// TIA Portal V17 export
// export: Created 2023-04-07T13:41:58.3192772Z, ExportSetting WithDefaults, DisplayName Totally Integrated Automation Portal, DisplayVersion V17 Update 4, DisplayName TIA Portal Openness, DisplayVersion V17 Update 4, DisplayName TIA Portal Version Control Interface, DisplayVersion V17, DisplayName STEP 7 Professional, DisplayVersion V17 Update 4, DisplayName STEP 7 Safety, DisplayVersion V17, DisplayName WinCC Professional, DisplayVersion V17 Update 4
VAR_GLOBAL   // PLC tag table "Tabella delle variabili standard"
   "M12.0_Paolo" AT %M12.0 : Bool;
   "M12.1_Paolo" AT %M12.1 : Bool;
   System_Byte AT %MB1 : Byte;
   FirstScan AT %M1.0 : Bool;
   DiagStatusUpdate AT %M1.1 : Bool;
   AlwaysTRUE AT %M1.2 : Bool;
   AlwaysFALSE AT %M1.3 : Bool;
   Clock_Byte AT %MB0 : Byte;
   Clock_10Hz AT %M0.0 : Bool;
   Clock_5Hz AT %M0.1 : Bool;
   "Clock_2.5Hz" AT %M0.2 : Bool;
   Clock_2Hz AT %M0.3 : Bool;
   "Clock_1.25Hz" AT %M0.4 : Bool;
   Clock_1Hz AT %M0.5 : Bool;
   "Clock_0.625Hz" AT %M0.6 : Bool;
   "Clock_0.5Hz" AT %M0.7 : Bool;
   xDxP1 AT %M104.0 : Bool;
   xDxP2 AT %M104.1 : Bool;
   xDxP3 AT %M104.2 : Bool;
   xDxP4 AT %M104.3 : Bool;
   xSxP1 AT %M105.0 : Bool;
   xSxP2 AT %M105.1 : Bool;
   xSxP3 AT %M105.2 : Bool;
   xSxP4 AT %M105.3 : Bool;
   xPE1P1 AT %M106.0 : Bool;
   xPE1P2 AT %M106.1 : Bool;
   xPE1P3 AT %M106.2 : Bool;
   xPE1P4 AT %M106.3 : Bool;
   xMVSP1 AT %M107.0 : Bool;
   xMVSP2 AT %M107.1 : Bool;
   xMVSP3 AT %M107.2 : Bool;
   xMVSP4 AT %M107.3 : Bool;
   xPlcRun AT %M2.0 : Bool;
   xAlwaysOff AT %M20.0 : Bool;
   xPEP1 AT %M108.0 : Bool;
   xPEP2 AT %M108.1 : Bool;
   xPEP3 AT %M108.2 : Bool;
   xPEP4 AT %M108.3 : Bool;
   xSM1P1 AT %M109.0 : Bool;
   xSM1P2 AT %M109.1 : Bool;
   xSM2P1 AT %M109.4 : Bool;
   xSM2P2 AT %M109.5 : Bool;
   xAckPS AT %M110.0 : Bool;
   xPE10P1 AT %M106.4 : Bool;
   xPE10P2 AT %M106.5 : Bool;
   xPE10P3 AT %M106.6 : Bool;
   xPE10P4 AT %M106.7 : Bool;
   xDx10P1 AT %M104.4 : Bool;
   xDx10P2 AT %M104.5 : Bool;
   xDx10P3 AT %M104.6 : Bool;
   xDx10P4 AT %M104.7 : Bool;
   xSx10P1 AT %M105.4 : Bool;
   xSx10P2 AT %M105.5 : Bool;
   xSx10P3 AT %M105.6 : Bool;
   xSx10P4 AT %M105.7 : Bool;
   xFPlocal AT %M110.4 : Bool;
   xPEP11 AT %M108.4 : Bool;
   xPEP21 AT %M108.5 : Bool;
   xPEP31 AT %M108.6 : Bool;
   xPEP41 AT %M108.7 : Bool;
   xFNlocal AT %M110.5 : Bool;
   xDPCATL1 AT %M120.0 : Bool;
   xDPCATL2 AT %M120.1 : Bool;
   xMVSP11 AT %M107.4 : Bool;
   xMVSP21 AT %M107.5 : Bool;
   xMVSP31 AT %M107.6 : Bool;
   xMVSP41 AT %M107.7 : Bool;
   xxxxxxxxxxxxxxxxxxxxxxxxxxxxxxxx AT %M100.0 : Bool;
   Tag_1 AT %M300.0 : Bool;
   Tag_2 AT %M300.1 : Bool;
   Tag_3 AT %M300.2 : Bool;
END_VAR
